{attribute 'qualified_only'}
TYPE enAccessLevel :
(
	logged_out,
	operator,
	maintenance,
	admin,
	help_tec,
	max_
);
END_TYPE

(* stored: Version 1.1.0.1, ProductVersion 3.1.4024.6
   DUT enAccessLevel: Id {56ee4e33-cdb0-44d0-b4bc-efc8a52a9aec} *)
